
FUNCTION CB_dint_to_word : WORD

TITLE = ' Convert a double integer into an word '
VERSION : '1.0'
AUTHOR  : CB
NAME    : DintToWo
FAMILY  : TNI

VAR_INPUT
    IN : DINT;
END_VAR

VAR_TEMP

END_VAR

BEGIN

CB_dint_to_word := DINT_TO_WORD(IN);

END_FUNCTION
